FUNCTION_BLOCK FB_XPlanarGamePad
VAR_IN_OUT
	fbMover							: MC_PlanarMover; //XPlanar Mover
	fbMoverAxis						: ARRAY [1..cuiMoverAxisSize] OF AXIS_REF; //ExternalSetPoint Axes 1-6:x,y,z,a,b,c
END_VAR
VAR_INPUT
	GamePad							: ST_GamePad; //The GamePad input
	XPlanarGamePadCondition			: ST_XPlanarGamePadCondition; //The moving Conditions
	KindMover						: uiKindMover := uiKindMover.AMP4330; //The mover kind. To limit tile.
	lrStickDeadZone					: LREAL := 10000; //The Stick DeadZone
	lrMinLimitPosX					: LREAL := 0; //XPlanar Tile limit min position X.
	lrMaxLimitPosX					: LREAL := 960; //XPlanar Tile limit max position X.
	lrMinLimitPosY					: LREAL := 0; //XPlanar Tile limit min position Y.
	lrMaxLimitPosY					: LREAL := 720; //XPlanar Tile limit max position Y.
END_VAR
VAR_OUTPUT
	stStatus						: uiStatus_XPGamePad; //FB status
END_VAR

VAR //checkgamepad
	afbR_Trig						: ARRAY [0..cuiGamePadSize] OF R_TRIG; //Check GamePad trigger
	abToggle						: ARRAY [0..cuiGamePadSize] OF BOOL; //A button trigger convert toggle. 
	abBusy							: ARRAY [0..cuiGamePadSize] OF BOOL; //A button command busy check.
	afbFeedback						: ARRAY [0..cuiGamePadSize] OF MC_PlanarFeedback;
END_VAR
VAR //command
	//General
	uiCommand						: UINT; //command method
	stActPos						: MoverVector;
	lrLimitFreeMove_AB				: LREAL := 1;
	stBasePos						: MoverVector;
	alrSetLimitPosMax				: ARRAY [0..1] OF LREAL;
	alrSetLimitPosMin				: ARRAY [0..1] OF LREAL;
	lrLimitBuffer					: LREAL := 5; 
	//Dpad
	stPosition_Dpad					: PositionXYC;
	stSetPos_Dpad					: MoverVector;
	stCondition_Dpad				: DynamicConstraint_PathXY;
	//LeftStickX
	afbMoveAbs_LeftStickX			: ARRAY [0..1] OF MC_MoveAbsolute;
	lrVelocity_LeftStickX			: LREAL;
	lrTempVelocity_LeftStickX		: LREAL;
	//LeftStickY
	afbMoveAbs_LeftStickY			: ARRAY [0..1] OF MC_MoveAbsolute;
	lrVelocity_LeftStickY			: LREAL;
	lrTempVelocity_LeftStickY		: LREAL;
	//RightStickX
	afbMoveAbs_RightStickX			: ARRAY [0..1] OF MC_MoveAbsolute;
	lrPosition_RightStickX			: LREAL;
	lrTempPosition_RightStickX		: LREAL;
	//RightStickY
	afbMoveAbs_RightStickY			: ARRAY [0..1] OF MC_MoveAbsolute;
	lrPosition_RightStickY			: LREAL;
	lrTempPosition_RightStickY		: LREAL;
	//ButtonA
	lrPosition_ButtonA				: LREAL;
	stCondition_ButtonA				: DynamicConstraint_PathXY;
	//ButtonY
	fbTon_ButtonY					: TON;
	fbTcRestart_ButtonY				: TC_Restart;
	//ButtonLR
	lrPosition_ButtonLR				: LREAL;
	stCondition_ButtonLR			: DynamicConstraint_Path;

	//Start
	afbPower						: ARRAY [1..cuiMoverAxisSize] OF MC_Power;
	bPowered						: BOOL; //Power
	//Select
	afbReset						: ARRAY [1..cuiMoverAxisSize] OF MC_Reset;
END_VAR
VAR //externalsetpoint
	stSetpoint_Pos					: MoverVector;
	stSetpoint_Vel					: MoverVector;
	stSetpoint_Acc					: MoverVector;
	stESGOptions					: ST_ExternalSetpointGenerationOptions;
END_VAR
VAR //FB
	uiIndex							: UINT;
END_VAR
VAR CONSTANT
	cuiLimitStick					: UINT := 32767;
	cuiMoverAxisSize				: UINT := 6;
	cuiGamePadSize					: UINT := 30;
	
END_VAR

//現在位置の更新
stActPos := fbMover.MCTOPLC.ACT.ActPos;
//動作限界の決定
alrSetLimitPosMax[0] := mCalculateLimitPosition(bDirection:= TRUE,lrLimitPosition:= lrMaxLimitPosX, KindMover:= KindMover) - lrLimitBuffer;
alrSetLimitPosMax[1] := mCalculateLimitPosition(bDirection:= TRUE,lrLimitPosition:= lrMaxLimitPosY, KindMover:= KindMover) - lrLimitBuffer;
alrSetLimitPosMin[0] := mCalculateLimitPosition(bDirection:= FALSE,lrLimitPosition:= lrMinLimitPosX, KindMover:= KindMover) + lrLimitBuffer;
alrSetLimitPosMin[1] := mCalculateLimitPosition(bDirection:= FALSE,lrLimitPosition:= lrMinLimitPosY, KindMover:= KindMover) + lrLimitBuffer;

//GamePadの入力確認と入力に対する動作の実行
mCheckGamePad();
//ExternalSetpointの処理
mExternalSetpoint();

FOR uiIndex:=0 TO cuiGamePadSize DO
	afbFeedback[uiIndex].Update();
END_FOR

METHOD PRIVATE mApplyDeadZone : LREAL
VAR_INPUT
	lrValue						: LREAL;
	lrDeadzone					: LREAL;
	lrMaxValue					: LREAL;
END_VAR
VAR
	lrAbsValue					: LREAL;
	lrOutput					: LREAL;
	lrScale						: LREAL;
END_VAR
lrAbsValue := ABS(lrValue);

IF lrAbsValue <= lrDeadzone THEN
	lrOutput := 0;
ELSE
	lrScale := lrMaxValue / (lrMaxValue - lrDeadzone);
	lrOutput := (lrAbsValue - lrDeadzone) * lrScale;
	
	//search minimum value among the argument
	lrOutput := MIN(lrOutput, lrMaxValue);
END_IF

IF lrValue < 0 THEN
	lrOutput := -lrOutput;
END_IF

mApplyDeadZone := lrOutput;
END_METHOD

METHOD PRIVATE mCalculateLimitAngle : LREAL
VAR_INPUT
	KindMover				: uiKindMover;
	z						: LREAL;
END_VAR
VAR
	lrMoverSize				: LREAL;
	stMoverSize				: ST_MoverSize;
END_VAR
IF KindMover = uiKindMover.AMP4220 THEN
	lrMoverSize := stMoverSize.AMP4220;
ELSIF KindMover = uiKindMover.AMP4550 THEN
	lrMoverSize := stMoverSize.AMP4550;
ELSE
	lrMoverSize := stMoverSize.AMP4330;
END_IF

mCalculateLimitAngle := ATAN(z/lrMoverSize) * (180.0/3.14);
END_METHOD

METHOD PRIVATE mCalculateLimitPosition : LREAL
VAR_INPUT
	bDirection						: BOOL; //0:Min 1:Max
	lrLimitPosition					: LREAL;
	KindMover						: uiKindMover;
END_VAR
VAR
	lrMoverSize				: LREAL;
	stMoverSize				: ST_MoverSize;
END_VAR
IF KindMover = uiKindMover.AMP4220 THEN
	lrMoverSize := stMoverSize.AMP4220;
ELSIF KindMover = uiKindMover.AMP4550 THEN
	lrMoverSize := stMoverSize.AMP4550;
ELSE
	lrMoverSize := stMoverSize.AMP4330;
END_IF

IF bDirection THEN
	mCalculateLimitPosition := lrLimitPosition - lrMoverSize/2;
ELSE
	mCalculateLimitPosition := lrLimitPosition + lrMoverSize/2;
END_IF
END_METHOD

METHOD PRIVATE mCheckGamePad : BOOL
VAR_INPUT
END_VAR
//ButtonSelect 
//Reset errors
afbR_Trig[uiGamePad.ButtonSelect](CLK:= GamePad.ButtonSelect, Q=> );
IF afbR_Trig[uiGamePad.ButtonSelect].Q THEN
	abToggle[uiGamePad.ButtonSelect] := NOT abToggle[uiGamePad.ButtonSelect];
END_IF
uiCommand := uiGamePad.ButtonSelect;
mCommand();
mCheckStatus();
IF THIS^.fbMover.MCTOPLC.STD.State = MC_PLANAR_STATE.Error THEN
	RETURN;
END_IF

//ButtonStart 
//Power
afbR_Trig[uiGamePad.ButtonStart](CLK:= GamePad.ButtonStart, Q=> );
IF afbR_Trig[uiGamePad.ButtonStart].Q THEN
	abToggle[uiGamePad.ButtonStart] := NOT abToggle[uiGamePad.ButtonStart];
END_IF
uiCommand := uiGamePad.ButtonStart;
mCommand();
mCheckStatus();
IF NOT THIS^.fbMover.MCTOPLC.STD.State = MC_PLANAR_STATE.Enabled THEN
	RETURN;
END_IF

//Virtual Axis PowerControll
//Pad
afbR_Trig[uiGamePad.DPadDown](CLK:= GamePad.DPadDown, Q=> );
afbR_Trig[uiGamePad.DPadLeft](CLK:= GamePad.DPadLeft, Q=> );
afbR_Trig[uiGamePad.DPadRight](CLK:= GamePad.DPadRight, Q=> );
afbR_Trig[uiGamePad.DPadUp](CLK:= GamePad.DPadUp, Q=> );
IF afbR_Trig[uiGamePad.DPadUp].Q
OR afbR_Trig[uiGamePad.DPadDown].Q
OR afbR_Trig[uiGamePad.DPadLeft].Q 
OR afbR_Trig[uiGamePad.DPadRight].Q THEN
	abToggle[uiGamePad.Dpad] := TRUE;
END_IF
uiCommand := uiGamePad.Dpad;
mCommand();
mCheckStatus();
//ButtonA 
//move z
afbR_Trig[uiGamePad.ButtonA](CLK:= GamePad.ButtonA, Q=> );
IF afbR_Trig[uiGamePad.ButtonA].Q THEN
	abToggle[uiGamePad.ButtonA] := NOT abToggle[uiGamePad.ButtonA];
END_IF
uiCommand := uiGamePad.ButtonA;
mCommand();
mCheckStatus();
//ButtonB
afbR_Trig[uiGamePad.ButtonB](CLK:= GamePad.ButtonB, Q=> );
IF afbR_Trig[uiGamePad.ButtonB].Q THEN
	abToggle[uiGamePad.ButtonB] := NOT abToggle[uiGamePad.ButtonB];
END_IF
uiCommand := uiGamePad.ButtonB;
mCommand();
mCheckStatus();
//ButtonX
afbR_Trig[uiGamePad.ButtonX](CLK:= GamePad.ButtonA, Q=> );
IF afbR_Trig[uiGamePad.ButtonX].Q THEN
	abToggle[uiGamePad.ButtonX] := NOT abToggle[uiGamePad.ButtonX];
END_IF
uiCommand := uiGamePad.ButtonX;
mCommand();
mCheckStatus();
//ButtonY
afbR_Trig[uiGamePad.ButtonY](CLK:= GamePad.ButtonY, Q=> );
IF afbR_Trig[uiGamePad.ButtonY].Q THEN
	abToggle[uiGamePad.ButtonY] := NOT abToggle[uiGamePad.ButtonY];
END_IF
uiCommand := uiGamePad.ButtonY;
mCommand();
mCheckStatus();
//Button L1 
//move C
afbR_Trig[uiGamePad.ButtonL1](CLK:= GamePad.ButtonL1, Q=> );
IF afbR_Trig[uiGamePad.ButtonL1].Q THEN
	abToggle[uiGamePad.ButtonL1] := NOT abToggle[uiGamePad.ButtonL1];
END_IF
afbR_Trig[uiGamePad.ButtonR1](CLK:= GamePad.ButtonR1, Q=> );
IF afbR_Trig[uiGamePad.ButtonR1].Q THEN
	abToggle[uiGamePad.ButtonR1] := NOT abToggle[uiGamePad.ButtonR1];
END_IF
afbR_Trig[uiGamePad.ButtonL2](CLK:= GamePad.ButtonL2, Q=> );
IF afbR_Trig[uiGamePad.ButtonL2].Q THEN
	abToggle[uiGamePad.ButtonL2] := NOT abToggle[uiGamePad.ButtonL2];
END_IF
afbR_Trig[uiGamePad.ButtonR2](CLK:= GamePad.ButtonR2, Q=> );
IF afbR_Trig[uiGamePad.ButtonR2].Q THEN
	abToggle[uiGamePad.ButtonR2] := NOT abToggle[uiGamePad.ButtonR2];
END_IF
IF afbR_Trig[uiGamePad.ButtonL1].Q 
OR afbR_Trig[uiGamePad.ButtonR1].Q 
OR afbR_Trig[uiGamePad.ButtonL2].Q 
OR afbR_Trig[uiGamePad.ButtonR2].Q THEN
	abToggle[uiGamePad.ButtonLR] := NOT abToggle[uiGamePad.ButtonLR];
END_IF
uiCommand := uiGamePad.ButtonLR;
mCommand();
mCheckStatus();
//Trigger L2
uiCommand := uiGamePad.TriggerL2;
mCommand();
mCheckStatus();
//Trigger R2
uiCommand := uiGamePad.TriggerR2;
mCommand();
mCheckStatus();
//LStick 
//move free XY
uiCommand := uiGamePad.LeftStickX;
mCommand();
mCheckStatus();
uiCommand := uiGamePad.LeftStickY;
mCommand();
mCheckStatus();

//RStick 
//move free AB
uiCommand := uiGamePad.RightStickX;
mCommand();
mCheckStatus();
uiCommand := uiGamePad.RightStickY;
mCommand();
mCheckStatus();
END_METHOD

METHOD PRIVATE mCheckStatus : uiStatus_XPGamePad
VAR_INPUT
END_VAR
IF abBusy[uiGamePad.Dpad] THEN
	stStatus := uiStatus_XPGamePad.MovingDpad;
ELSIF abBusy[uiGamePad.ButtonLR] THEN
	stStatus := uiStatus_XPGamePad.RotationC;
ELSIF TO_INT(stBasePos.x) <> TO_INT(stActPos.x) AND TO_INT(stBasePos.y) <> TO_INT(stActPos.y) THEN
	stStatus := uiStatus_XPGamePad.CantRotationC;
ELSIF bPowered THEN
	stStatus := uiStatus_XPGamePad.Ready;
ELSE
	stStatus := uiStatus_XPGamePad.Disable;
END_IF
END_METHOD

METHOD PRIVATE mCommand : BOOL
VAR_INPUT
END_VAR
VAR
	i								: UINT;
	stCondition_: INT;
	lrValue_Stick : LREAL;
	lrSetTargetPosition : LREAL;
END_VAR
CASE uiCommand OF
uiGamePad.Dpad: //Move the position that a Mover can rotate C
	//Cant move until moving XY
	IF stStatus = uiStatus_XPGamePad.RotationC THEN
		abToggle[uiGamePad.Dpad] := FALSE;
		RETURN;
	END_IF
		
	IF abToggle[uiGamePad.Dpad] AND NOT abBusy[uiGamePad.Dpad] THEN
		//The set position to move
		//The set position dont be set opposite direction
		IF afbR_Trig[uiGamePad.DPadRight].Q AND alrSetLimitPosMax[0] > stBasePos.x + 120 THEN
			stBasePos.x := stBasePos.x + 120;	
		ELSIF afbR_Trig[uiGamePad.DPadLeft].Q AND alrSetLimitPosMin[0] < stBasePos.x - 120 THEN
			stBasePos.x := stBasePos.x - 120;
		END_IF
		IF afbR_Trig[uiGamePad.DPadUp].Q AND alrSetLimitPosMax[1] > stBasePos.y + 120 THEN
			stBasePos.y := stBasePos.y + 120;
		ELSIF afbR_Trig[uiGamePad.DPadDown].Q AND alrSetLimitPosMin[1] < stBasePos.y - 120 THEN
			stBasePos.y := stBasePos.y - 120;
		END_IF
		stSetPos_Dpad.x := stBasePos.x;
		stSetPos_Dpad.y := stBasePos.y;
		//Set Position and move condition
		stPosition_Dpad.SetValuesXYC(
			x:= stSetPos_Dpad.x, y:= stSetPos_Dpad.y, c:= stSetPos_Dpad.c
		);
		stCondition_Dpad.SetValuesVADJ(
			V:= XPlanarGamePadCondition.lrVelocity_ABC, A:= XPlanarGamePadCondition.lrAcceleration_ABC, 
			D:= XPlanarGamePadCondition.lrDeceleration_ABC, J:= XPlanarGamePadCondition.lrJerk_ABC
		);
		//A mover is operated to move with XY planar
		fbMover.MoveToPosition(
			 commandFeedback:= afbFeedback[uiGamePad.Dpad],
			 targetPosition:= stPosition_Dpad,
			 constraint:= stCondition_Dpad,
			 options:= 0
		);
		//check moving
		abBusy[uiGamePad.Dpad] := TRUE;
	ELSE
		//Check a mover finished moving
		IF NOT afbFeedback[uiGamePad.Dpad].Active THEN
			abBusy[uiGamePad.Dpad] := FALSE;
			abToggle[uiGamePad.DPadDown] := FALSE;
			abToggle[uiGamePad.DPadLeft] := FALSE;
			abToggle[uiGamePad.DPadRight] := FALSE;
			abToggle[uiGamePad.DPadUp] := FALSE;
			abToggle[uiGamePad.Dpad] := FALSE;
		END_IF
	END_IF
		
uiGamePad.LeftStickX: //A mover move in the x direction with externalsetpoint
	IF stStatus = uiStatus_XPGamePad.RotationC THEN
		RETURN;
	END_IF
	//Record a previous set position
	lrTempVelocity_LeftStickX := lrVelocity_LeftStickX;
	//Calculate to correct Lstick
	lrValue_Stick := mApplyDeadZone
					(
						lrValue:= TO_LREAL(GamePad.LeftStickX),
						lrDeadzone:= lrStickDeadzone, 
						lrMaxValue:= TO_LREAL(cuiLimitStick)
					);
	lrVelocity_LeftStickX := XPlanarGamePadCondition.lrVelocity_XYZ * (lrValue_Stick / TO_LREAL(cuiLimitStick));
	IF lrVelocity_LeftStickX > 0 THEN
		//最大エリア範囲を設定
		lrSetTargetPosition := alrSetLimitPosMax[0] - stBasePos.x;
	ELSIF lrVelocity_LeftStickX < 0 THEN
		//最小エリア範囲を設定
		lrSetTargetPosition := alrSetLimitPosMin[0] - stBasePos.x;
	ELSE
		lrSetTargetPosition := 0;
		lrVelocity_LeftStickX := XPlanarGamePadCondition.lrVelocity_XYZ /2;
	END_IF
	//Alternate orders to MC_MoveAbsolute
	IF lrTempVelocity_LeftStickX <> lrVelocity_LeftStickX THEN
		IF (NOT afbMoveAbs_LeftStickX[0].busy AND NOT afbMoveAbs_LeftStickX[1].busy) 
		OR (NOT afbMoveAbs_LeftStickX[0].busy AND afbMoveAbs_LeftStickX[1].busy) THEN
			afbMoveAbs_LeftStickX[0].Execute := TRUE;
			afbMoveAbs_LeftStickX[1].Execute := FALSE;
		ELSIF (afbMoveAbs_LeftStickX[0].busy AND NOT afbMoveAbs_LeftStickX[1].busy) THEN
			afbMoveAbs_LeftStickX[0].Execute := FALSE;
			afbMoveAbs_LeftStickX[1].Execute := TRUE;
		END_IF 
	END_IF
	FOR i:=0 TO 1 DO
		afbMoveAbs_LeftStickX[i]
		(
			Axis:= fbMoverAxis[1],
			Position:= lrSetTargetPosition, 
			Velocity:= ABS(lrVelocity_LeftStickX), 
			Acceleration:= XPlanarGamePadCondition.lrAcceleration_XYZ, 
			Deceleration:= XPlanarGamePadCondition.lrDeceleration_XYZ, 
			Jerk:= XPlanarGamePadCondition.lrJerk_XYZ
		);
		afbMoveAbs_LeftStickX[i].Execute := FALSE;
	END_FOR

uiGamePad.LeftStickY: //A mover move in the Y direction with externalsetpoint
	IF stStatus = uiStatus_XPGamePad.RotationC THEN
		RETURN;
	END_IF
	//Same logic as LeftStickX
	lrTempVelocity_LeftStickY := lrVelocity_LeftStickY;
	lrValue_Stick := mApplyDeadZone
					(
						lrValue:= TO_LREAL(GamePad.LeftStickY),
						lrDeadzone:= lrStickDeadzone, 
						lrMaxValue:= TO_LREAL(cuiLimitStick)
					);
	lrVelocity_LeftStickY := XPlanarGamePadCondition.lrVelocity_XYZ * (lrValue_Stick / TO_LREAL(cuiLimitStick)); 
	IF lrVelocity_LeftStickY > 0 THEN
		//最大エリア範囲を設定
		lrSetTargetPosition := alrSetLimitPosMax[1] - stBasePos.y;
	ELSIF lrVelocity_LeftStickY < 0 THEN
		//最小エリア範囲を設定
		lrSetTargetPosition := alrSetLimitPosMin[1] - stBasePos.y;
	ELSE
		lrSetTargetPosition := 0;
		lrVelocity_LeftStickY := XPlanarGamePadCondition.lrVelocity_XYZ /2;
	END_IF
	IF lrTempVelocity_LeftStickY <> lrVelocity_LeftStickY THEN
		IF (NOT afbMoveAbs_LeftStickY[0].busy AND NOT afbMoveAbs_LeftStickY[1].busy) 
		OR (NOT afbMoveAbs_LeftStickY[0].busy AND afbMoveAbs_LeftStickY[1].busy) THEN
			afbMoveAbs_LeftStickY[0].Execute := TRUE;
			afbMoveAbs_LeftStickY[1].Execute := FALSE;
		ELSIF (afbMoveAbs_LeftStickY[0].busy AND NOT afbMoveAbs_LeftStickY[1].busy) THEN
			afbMoveAbs_LeftStickY[0].Execute := FALSE;
			afbMoveAbs_LeftStickY[1].Execute := TRUE;
		END_IF 
	END_IF
	FOR i:=0 TO 1 DO
		afbMoveAbs_LeftStickY[i]
		(
			Axis:= fbMoverAxis[2],
			Position:= lrSetTargetPosition, 
			Velocity:= ABS(lrVelocity_LeftStickY), 
			Acceleration:= XPlanarGamePadCondition.lrAcceleration_XYZ, 
			Deceleration:= XPlanarGamePadCondition.lrDeceleration_XYZ, 
			Jerk:= XPlanarGamePadCondition.lrJerk_XYZ
		);
		afbMoveAbs_LeftStickY[i].Execute := FALSE;
	END_FOR

uiGamePad.RightStickX: //AB free move
	//Same Logic as LStick
	//Calculate the values of the limit according to Z value.
	lrLimitFreeMove_AB := mCalculateLimitAngle(KindMover:= KindMover, z:= stActPos.z);
	lrTempPosition_RightStickX := lrPosition_RightStickX;
	lrValue_Stick := mApplyDeadZone
					(
						lrValue:= TO_LREAL(GamePad.RightStickX),
						lrDeadzone:= lrStickDeadzone, 
						lrMaxValue:= TO_LREAL(cuiLimitStick)
					);
	lrPosition_RightStickX := lrLimitFreeMove_AB * (lrValue_Stick / TO_LREAL(cuiLimitStick));
	IF lrTempPosition_RightStickX <> lrPosition_RightStickX THEN
		IF (NOT afbMoveAbs_RightStickX[0].busy AND NOT afbMoveAbs_RightStickX[1].busy) 
		OR (NOT afbMoveAbs_RightStickX[0].busy AND afbMoveAbs_RightStickX[1].busy) THEN
			afbMoveAbs_RightStickX[0].Execute := TRUE;
			afbMoveAbs_RightStickX[1].Execute := FALSE;
		ELSIF (afbMoveAbs_RightStickX[0].busy AND NOT afbMoveAbs_RightStickX[1].busy) THEN
			afbMoveAbs_RightStickX[0].Execute := FALSE;
			afbMoveAbs_RightStickX[1].Execute := TRUE;
		END_IF 
	END_IF
	FOR i:=0 TO 1 DO
		afbMoveAbs_RightStickX[i]
		(
			Axis:= fbMoverAxis[5],
			Position:= lrPosition_RightStickX, 
			Velocity:= XPlanarGamePadCondition.lrVelocity_ABC, 
			Acceleration:= XPlanarGamePadCondition.lrAcceleration_ABC, 
			Deceleration:= XPlanarGamePadCondition.lrDeceleration_ABC, 
			Jerk:= XPlanarGamePadCondition.lrJerk_ABC
		);
		afbMoveAbs_RightStickX[i].Execute := FALSE;
	END_FOR
	
uiGamePad.RightStickY: //AB free move
	//Same logic as RightStickX

	lrLimitFreeMove_AB := mCalculateLimitAngle(KindMover:= KindMover, z:= stActPos.z);
	lrTempPosition_RightStickY := lrPosition_RightStickY;
	lrValue_Stick := mApplyDeadZone
					(
						lrValue:= TO_LREAL(GamePad.RightStickY),
						lrDeadzone:= lrStickDeadzone, 
						lrMaxValue:= TO_LREAL(cuiLimitStick)
					);
	lrPosition_RightStickY := lrLimitFreeMove_AB * (lrValue_Stick / UINT_TO_LREAL(cuiLimitStick));
	IF lrTempPosition_RightStickY <> lrPosition_RightStickY THEN
		IF (NOT afbMoveAbs_RightStickY[0].busy AND NOT afbMoveAbs_RightStickY[1].busy) 
		OR (NOT afbMoveAbs_RightStickY[0].busy AND afbMoveAbs_RightStickY[1].busy) THEN
			afbMoveAbs_RightStickY[0].Execute := TRUE;
			afbMoveAbs_RightStickY[1].Execute := FALSE;
		ELSIF (afbMoveAbs_RightStickY[0].busy AND NOT afbMoveAbs_RightStickY[1].busy) THEN
			afbMoveAbs_RightStickY[0].Execute := FALSE;
			afbMoveAbs_RightStickY[1].Execute := TRUE;
		END_IF 
	END_IF
	FOR i:=0 TO 1 DO
		afbMoveAbs_RightStickY[i]
		(
			Axis:= fbMoverAxis[4],
			Position:= -lrPosition_RightStickY, 
			Velocity:= XPlanarGamePadCondition.lrVelocity_ABC, 
			Acceleration:= XPlanarGamePadCondition.lrAcceleration_ABC, 
			Deceleration:= XPlanarGamePadCondition.lrDeceleration_ABC, 
			Jerk:= XPlanarGamePadCondition.lrJerk_ABC
		);
		afbMoveAbs_RightStickY[i].Execute := FALSE;
	END_FOR
	
uiGamePad.ButtonA: //A mover up to z direction
IF abToggle[uiGamePad.ButtonA] AND NOT abBusy[uiGamePad.ButtonA] THEN
	IF stActPos.z > 3 THEN
		lrPosition_ButtonA := 2.0;
	ELSE
		lrPosition_ButtonA := 5.0;
	END_IF
	stCondition_ButtonA.SetValuesVADJ(
		V:= XPlanarGamePadCondition.lrVelocity_XYZ, A:= XPlanarGamePadCondition.lrAcceleration_XYZ, 
		D:= XPlanarGamePadCondition.lrDeceleration_XYZ, J:= XPlanarGamePadCondition.lrJerk_XYZ
	);
	fbMover.MoveZ(
		commandFeedback:= afbFeedback[uiGamePad.ButtonA], 
		targetPosition:= lrPosition_ButtonA, 
		constraint:= stCondition_ButtonA
	);
	abBusy[uiGamePad.ButtonA] := TRUE;
ELSE
	IF NOT afbFeedback[uiGamePad.ButtonA].Active THEN
		abBusy[uiGamePad.ButtonA] := FALSE;
		abToggle[uiGamePad.ButtonA] := FALSE;
	END_IF
END_IF

uiGamePad.ButtonB:
	//Reserve

uiGamePad.ButtonX:
	//Reserve
	
uiGamePad.ButtonY:
	//Reserve
IF abToggle[uiGamePad.ButtonY] THEN
	fbTon_ButtonY(IN:= TRUE, PT:= T#5S, Q=> , ET=> );
	IF fbTon_ButtonY.Q THEN
		fbTcRestart_ButtonY(
			NETID:= , 
			RESTART:= TRUE, 
			TMOUT:= , 
			BUSY=> , 
			ERR=> , 
			ERRID=> );
	END_IF
ELSE
	fbTon_ButtonY(IN:= FALSE, PT:= T#5S, Q=> , ET=> );
END_IF
	
	
	 
uiGamePad.ButtonLR:
	//Cant move until moving XY
	IF stStatus = uiStatus_XPGamePad.MovingDpad 
	OR stStatus = uiStatus_XPGamePad.CantRotationC THEN
		abToggle[uiGamePad.ButtonLR] := FALSE;
		RETURN;
	END_IF
	
	IF abToggle[uiGamePad.ButtonLR] AND NOT abBusy[uiGamePad.ButtonLR] THEN
		IF abToggle[uiGamePad.ButtonL1] THEN
			stBasePos.c := stBasePos.c + 90;
		ELSIF abToggle[uiGamePad.ButtonR1] THEN
			stBasePos.c := stBasePos.c - 90;
		ELSIF abToggle[uiGamePad.ButtonL2] THEN
			stBasePos.c := stBasePos.c + 360;
		ELSIF abToggle[uiGamePad.ButtonR2] THEN
			stBasePos.c := stBasePos.c - 360;
		END_IF
		lrPosition_ButtonLR := stBasePos.c;
		stCondition_ButtonLR.V := XPlanarGamePadCondition.lrVelocity_ABC;
		stCondition_ButtonLR.A := XPlanarGamePadCondition.lrAcceleration_ABC;
		stCondition_ButtonLR.D := XPlanarGamePadCondition.lrDeceleration_ABC;
		stCondition_ButtonLR.J := XPlanarGamePadCondition.lrJerk_ABC;
		fbMover.MoveC(
			commandFeedback:= afbFeedback[uiGamePad.ButtonLR], 
			targetPosition:= lrPosition_ButtonLR, 
			constraint:= stCondition_ButtonLR, 
			options:= 0
		);
		abBusy[uiGamePad.ButtonLR] := TRUE;
	ELSE
		IF NOT afbFeedback[uiGamePad.ButtonLR].Active THEN
			abBusy[uiGamePad.ButtonLR] := FALSE;
			abToggle[uiGamePad.ButtonL1] := FALSE;
			abToggle[uiGamePad.ButtonR1] := FALSE;
			abToggle[uiGamePad.ButtonL2] := FALSE;
			abToggle[uiGamePad.ButtonR2] := FALSE;
			abToggle[uiGamePad.ButtonLR] := FALSE;
		END_IF
	END_IF


uiGamePad.TriggerL2:
	//Reserve
	
uiGamePad.TriggerR2:
	//Reserve
	
uiGamePad.ButtonStart:
	//Power Control XPlanar
	IF abToggle[uiGamePad.ButtonStart] AND bPowered THEN
		fbMover.Disable(commandFeedback:= afbFeedback[uiGamePad.ButtonStart]);
		IF fbMover.MCTOPLC.STD.State = MC_PLANAR_STATE.Disabled THEN
			abToggle[uiGamePad.ButtonStart] := FALSE;
			bPowered := FALSE;
			abToggle[uiGamePad.ButtonStart] := FALSE;
			stStatus := uiStatus_XPGamePad.Disable;
		END_IF
	ELSIF abToggle[uiGamePad.ButtonStart] AND NOT bPowered THEN
		fbMover.Enable(commandFeedback:= afbFeedback[uiGamePad.ButtonStart]);
		IF fbMover.MCTOPLC.STD.State = MC_PLANAR_STATE.Enabled THEN
			abToggle[uiGamePad.ButtonStart] := FALSE;
			bPowered := TRUE;
			abToggle[uiGamePad.ButtonStart] := FALSE;
			stBasePos.x := XPlanarGamePadCondition.lrBasePosition_X;
			stBasePos.y := XPlanarGamePadCondition.lrBasePosition_X;
		END_IF
	END_IF
	//Power control ExternalSetpoint Axis
	IF bPowered THEN
		FOR i:=1 TO cuiMoverAxisSize DO
			afbPower[i].Enable := TRUE;
			afbPower[i].Enable_Negative := TRUE;
			afbPower[i].Enable_Positive := TRUE;
			afbPower[i](Axis:=fbMoverAxis[i]);
		END_FOR
	ELSE
		FOR i:=1 TO cuiMoverAxisSize DO
			afbPower[i].Enable := FALSE;
			afbPower[i].Enable_Negative := TRUE;
			afbPower[i].Enable_Positive := TRUE;
			afbPower[i](Axis:=fbMoverAxis[i]);
		END_FOR
	END_IF

uiGamePad.ButtonSelect:
	IF abToggle[uiGamePad.ButtonSelect] AND NOT abBusy[uiGamePad.ButtonSelect] THEN
		fbMover.Reset(commandFeedback:= afbFeedback[uiGamePad.ButtonSelect]);
		abBusy[uiGamePad.ButtonSelect] := TRUE;
		//ExternalSetPoint Axis error reset
		FOR i:=1 TO cuiMoverAxisSize DO
			afbReset[i].Execute := TRUE;
			afbReset[i](Axis:= fbMoverAxis[i]);
		END_FOR
	ELSE
		FOR i:=1 TO cuiMoverAxisSize DO
			afbReset[i].Execute := FALSE;
			afbReset[i](Axis:= fbMoverAxis[i]);
		END_FOR
		IF NOT afbFeedback[uiGamePad.ButtonSelect].Active THEN
			abBusy[uiGamePad.ButtonSelect] := FALSE;
			abToggle[uiGamePad.ButtonSelect] := FALSE;
		END_IF
	END_IF
	
END_CASE
END_METHOD

METHOD PRIVATE mExternalSetpoint : BOOL
VAR_INPUT
END_VAR
stSetpoint_Pos.x := fbMoverAxis[1].NcToPlc.ActPos;
stSetpoint_Pos.y := fbMoverAxis[2].NcToPlc.ActPos;
stSetpoint_Pos.z := fbMoverAxis[3].NcToPlc.ActPos;
stSetpoint_Pos.a := fbMoverAxis[4].NcToPlc.ActPos;
stSetpoint_Pos.b := fbMoverAxis[5].NcToPlc.ActPos;
stSetpoint_Pos.c := fbMoverAxis[6].NcToPlc.ActPos;

stSetpoint_Vel.x := fbMoverAxis[1].NcToPlc.ActVelo;
stSetpoint_Vel.y := fbMoverAxis[2].NcToPlc.ActVelo;
stSetpoint_Vel.z := fbMoverAxis[3].NcToPlc.ActVelo;
stSetpoint_Vel.a := fbMoverAxis[4].NcToPlc.ActVelo;
stSetpoint_Vel.b := fbMoverAxis[5].NcToPlc.ActVelo;
stSetpoint_Vel.c := fbMoverAxis[6].NcToPlc.ActVelo;

stSetpoint_Acc.x := fbMoverAxis[1].NcToPlc.ActAcc;
stSetpoint_Acc.y := fbMoverAxis[2].NcToPlc.ActAcc;
stSetpoint_Acc.z := fbMoverAxis[3].NcToPlc.ActAcc;
stSetpoint_Acc.a := fbMoverAxis[4].NcToPlc.ActAcc;
stSetpoint_Acc.b := fbMoverAxis[5].NcToPlc.ActAcc;
stSetpoint_Acc.c := fbMoverAxis[6].NcToPlc.ActAcc;
	
IF bPowered AND fbMover.MCTOPLC.STD.State = MC_PLANAR_STATE.Enabled THEN
	fbMover.SetExternalSetpoint(
		setPosition:= stSetpoint_Pos, 
		setVelocity:= stSetpoint_Vel, 
		setAcceleration:= stSetpoint_Acc);
	stESGOptions.mode := MC_EXTERNAL_SET_POSITION_MODE.Relative;
	fbMover.StartExternalSetpointGeneration(commandFeedback:= 0, options:= stESGOptions);
ELSE
	fbMover.StopExternalSetpointGeneration(commandFeedback:= 0);
END_IF
END_METHOD

END_FUNCTION_BLOCK

(* stored: Version 1.1.0.1
   POU FB_XPlanarGamePad: Id {d9dfe6f5-63c0-40ac-8f62-57f7720f7ddc}, SpecialFunc None
   Method mApplyDeadZone: Id {29817e3b-1c05-4160-8930-83a6636fa372}
   Method mCalculateLimitAngle: Id {ec5ed99d-04a0-4e57-9582-3139520850f0}
   Method mCalculateLimitPosition: Id {02d20284-81bc-4ddc-8c5f-603f4de60f5b}
   Method mCheckGamePad: Id {cd5a66b7-8bbf-4285-b3c0-dd4d583b4717}
   Method mCheckStatus: Id {7d50fac8-4fda-4e65-b65e-914dea797f8f}
   Method mCommand: Id {018a0f5d-cb2a-42ce-bd53-fb944e60cfc0}
   Method mExternalSetpoint: Id {707025e5-e543-4333-9a26-405e4c5c21e0} *)
